///EL1262 | XFC, 2-channel digital input terminal with oversampling
FUNCTION_BLOCK EL1262_v0_00

END_FUNCTION_BLOCK

(* stored: Version 1.1.0.1, ProductVersion 3.1.4022.6
   POU EL1262_v0_00: Id {71013e38-8a84-41a1-8711-92d41ae9502b}, SpecialFunc None *)
